PROGRAM PMPS
VAR
    
    fbArbiterIO : FB_SubSysToArbiter_IO;
END_VAR

fbArbiterIO(Arbiter := GVL.g_fbArbiter1, fbFFHWO := GVL.g_FastFaultOutput1);

END_PROGRAM

(* stored: Version 1.1.0.1, ProductVersion 3.1.4022.18
   POU PMPS: Id {9f17630a-fcaa-08bb-22bb-9b109c090d19}, SpecialFunc None *)
